// TIA Portal project "Examen_1" (V16)

(* hardware
DEVICE "S7-1200 station_1"  S7-1200 Station
   slot 0: "Rack_0"  S7-1200 Rack  Rack  V1.0
   slot 1: "PLC_1"  CPU 1215C DC/DC/DC  6ES7 215-1AG40-0XB0  V4.4
   slot 2: "AI 4x13BIT/AQ 2x14BIT_1"  SM 1234 AI4/AQ2  6ES7 234-4HE30-0XB0  V1.0
   slot 3: "AQ 1x12BIT_1"  AQ1 signal board  6ES7 232-4HA30-0XB0  V1.0
DEVICE "PC-System_1"  SIMATIC PC station
   slot 0: "Estación PC SIMATIC"  Rail  SIMATIC PC-Station  V1.0
      slot 125: "Stationmanager"  Station_Manager  V6.0.4
   slot 1: "HMI_RT_1"  WinCC RT Advanced  6AV2 104-0xxxx-xxxx  16.0.0.0
      slot 33792: "Interfaz del equipo"  Host interface
   slot 2: "IE general_1"  IE General  IE_CP  V8.2.0
*)

// ===== PLC "PLC_1"  CPU 1215C DC/DC/DC =====

VAR_GLOBAL   // PLC tag table "Tabla de variables estándar"
   "temp1_raw" AT %IW98 : Word;
   "temp2_raw" AT %IW66 : Word;
   "analog_out1" AT %QW80 : Word;
   "digital_out1" AT %Q0.0 : Bool;
END_VAR

DATA_BLOCK "Variables"   // DB1
{ S7_Optimized_Access := 'TRUE' }
VERSION : 0.1
   VAR
      temp1_norm : Real;
      temp1 : Real;
      temp2_norm : Real;
      temp2 : Real;
      out1_norm : Real;
      out1 : Real;
      out1_raw : Int;
      scada_pot : Int;
      scada_hour : Int;
      real_time : DTL;
      dtl_error : Int;
   END_VAR
BEGIN
END_DATA_BLOCK

ORGANIZATION_BLOCK "Main"   // OB1, LAD, ProgramCycle
TITLE = "Main Program Sweep (Cycle)"
{ S7_Optimized_Access := 'TRUE' }
VERSION : 0.1
   VAR_INPUT
      Initial_Call : Bool;   // Initial call of this OB
      Remanence : Bool;   // =True, if remanent data are available
   END_VAR
BEGIN

REGION Network 1 (SCL): Control de la salida analógica Q80
   // Si la hora introducida por SCADA coincide con la real, activar la salida Q0.0 y obtener 0V en la salida analógica QW80.
   // Si no se cumple la anterior condición, desactivar la salida Q0.0 y, si la temperatura 1 es menor a la temperatura 2, obtener 5V en la salida analógica QW80. De lo contrario, que dicha salida varie de -10 a 10V en función del potenciómetro en SCADA.
   IF "Variables".real_time.HOUR = "Variables".scada_hour THEN
       "Variables".out1_raw := 50;
       "digital_out1" := 1;
   ELSE
       "digital_out1" := 0;
       IF "Variables".temp1 < "Variables".temp2 THEN
           "Variables".out1_raw := 75;
       ELSE
           "Variables".out1_raw := "Variables".scada_pot;
       END_IF;
   END_IF;
END_REGION

REGION Network 2: Obtención del tiempo
   // Obtener la fecha y hora real y guardarla en una variable.
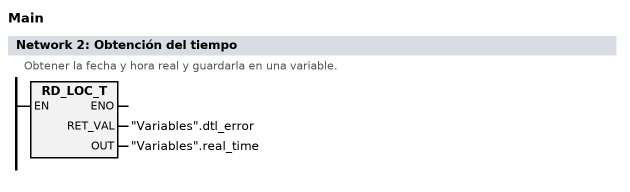
   "Variables".dtl_error := RD_LOC_T(OUT => "Variables".real_time);
END_REGION
END_ORGANIZATION_BLOCK

ORGANIZATION_BLOCK "Scales"   // OB123, LAD, ProgramCycle
TITLE = "Main Program Sweep (Cycle)"
{ S7_Optimized_Access := 'TRUE' }
VERSION : 0.1
   VAR_INPUT
      Initial_Call : Bool;   // Initial call of this OB
      Remanence : Bool;   // =True, if remanent data are available
   END_VAR
BEGIN

REGION Network 1: Escalado de la entrada analógica IW98
   // Escalado de un sensor de temperatura con salida 4..20mA para un rango de 20 a 100ºC.
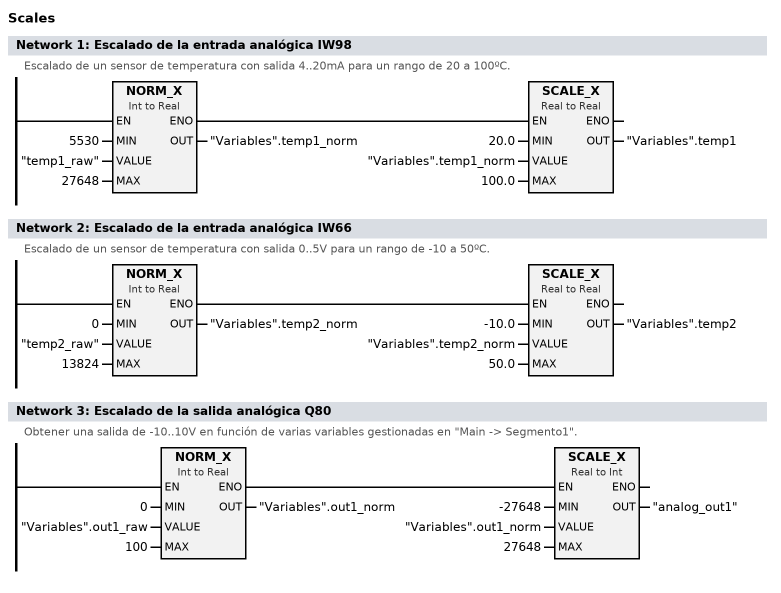
   RUNG wire#powerrail
      { S7_Templates := "[SrcType := Int, DestType := Real]" } Normalize(min := 5530, value := "temp1_raw", max := 27648, out => "Variables".temp1_norm)
      { S7_Templates := "[SrcType := Real, DestType := Real]" } Scale(min := 20.0, value := "Variables".temp1_norm, max := 100.0, out => "Variables".temp1)
   END_RUNG
   // the same network as SCL:
   "Variables".temp1_norm := NORM_X(MIN := 5530, VALUE := "temp1_raw", MAX := 27648);
   "Variables".temp1 := SCALE_X(MIN := 20.0, VALUE := "Variables".temp1_norm, MAX := 100.0);
END_REGION

REGION Network 2: Escalado de la entrada analógica IW66
   // Escalado de un sensor de temperatura con salida 0..5V para un rango de -10 a 50ºC.
   RUNG wire#powerrail
      { S7_Templates := "[SrcType := Int, DestType := Real]" } Normalize(min := 0, value := "temp2_raw", max := 13824, out => "Variables".temp2_norm)
      { S7_Templates := "[SrcType := Real, DestType := Real]" } Scale(min := -10.0, value := "Variables".temp2_norm, max := 50.0, out => "Variables".temp2)
   END_RUNG
   // the same network as SCL:
   "Variables".temp2_norm := NORM_X(MIN := 0, VALUE := "temp2_raw", MAX := 13824);
   "Variables".temp2 := SCALE_X(MIN := -10.0, VALUE := "Variables".temp2_norm, MAX := 50.0);
END_REGION

REGION Network 3: Escalado de la salida analógica Q80
   // Obtener una salida de -10..10V en función de varias variables gestionadas en "Main -> Segmento1".
   RUNG wire#powerrail
      { S7_Templates := "[SrcType := Int, DestType := Real]" } Normalize(min := 0, value := "Variables".out1_raw, max := 100, out => "Variables".out1_norm)
      { S7_Templates := "[SrcType := Real, DestType := Int]" } Scale(min := -27648, value := "Variables".out1_norm, max := 27648, out => "analog_out1")
   END_RUNG
   // the same network as SCL:
   "Variables".out1_norm := NORM_X(MIN := 0, VALUE := "Variables".out1_raw, MAX := 100);
   "analog_out1" := SCALE_X(MIN := -27648, VALUE := "Variables".out1_norm, MAX := 27648);
END_REGION
END_ORGANIZATION_BLOCK

(* ===== HMI "HMI_RT_1" =====
connection "HMI_Conexión_1": ETHERNET, S7_1200_OMS

HMI tags "Tabla de variables estándar"
   "Variables_temp1" : Real = PLC Variables.temp1, 1 s
   "Variables_temp2" : Real = PLC Variables.temp2, 1 s
   "Variables_scada_pot" : Int = PLC Variables.scada_pot, 1 s
   "Variables_real_time_HOUR" : USInt = PLC Variables.real_time.HOUR, 1 s
   "Variables_scada_hour" : Int = PLC Variables.scada_hour, 1 s

screen "Imagen_1" 800x600
   IOField "Campo ES_1" at 256,71 size 89x32; FormatPattern 999.9; Unit ºC
      ProcessValue <- "Variables_temp1"
   TextField "Campo de texto_1" at 274,37 size 76x22; Text 'Temp1'
   IOField "Campo ES_2" at 376,71 size 88x32; FormatPattern 999.9; Unit ºC
      ProcessValue <- "Variables_temp2"
   TextField "Campo de texto_2" at 393,37 size 76x22; Text 'Temp2'
   Slider "Deslizador_1" at 322,141 size 80x230; Caption 'SIMATIC'
      ProcessValue <- "Variables_scada_pot"
   IOField "Campo ES_3" at 274,445 size 64x32; FormatPattern 99
      ProcessValue <- "Variables_real_time_HOUR"
   TextField "Campo de texto_3" at 266,409 size 107x22; Text 'Real Hour'
   IOField "Campo ES_4" at 393,445 size 64x32; FormatPattern 99
      ProcessValue <- "Variables_scada_hour"
   TextField "Campo de texto_4" at 377,411 size 147x22; Text 'SCADA Hour'
*)